(* LS Electric XG5000 project: 241007_실습1PITA펑션제작 *)
(* PLC LSPLC *)

FUNCTION PITA : REAL
VAR_INPUT
    A변 : REAL;
    B변 : REAL;
END_VAR
VAR
    A2 : REAL;
    B2 : REAL;
    C2 : REAL;
    C변 : REAL;
END_VAR

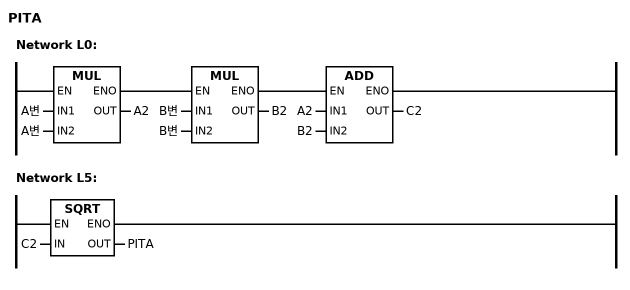
(* Rung L0 *)
A2 := A변 * A변;
B2 := B변 * B변;
C2 := A2 + B2;
(* Rung L5 *)
PITA := SQRT(C2);
END_FUNCTION

PROGRAM NewProgram (* task: 스캔 프로그램 *)
VAR
    Result : REAL;
    버튼 AT %IX0.0.0 : BOOL;
END_VAR

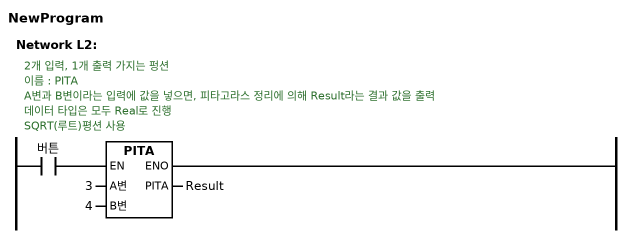
(* 2개 입력, 1개 출력 가지는 펑션 / 이름 : PITA / A변과 B변이라는 입력에 값을 넣으면, 피타고라스 정리에 의해 Result라는 결과 값을 출력 / 데이터 타입은 모두 Real로 진행 / SQRT(루트)평션 사용 *)
(* Rung L2 *)
IF 버튼 THEN Result := PITA(A변 := 3, B변 := 4); END_IF;
END_PROGRAM